FUNCTION_BLOCK BasicControlTS5 (* Basic Function Block Type *)
  (* Standard: 61499-2 *)
  (* Version 0.0, 6/17/2016, Andrei, nxtControl GmbH, Template *)
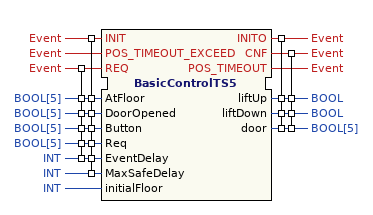
  EVENT_INPUT
    INIT WITH AtFloor, DoorOpened, Button, Req, EventDelay, MaxSafeDelay; (* Initialization Request *)
    POS_TIMEOUT_EXCEED;
    REQ WITH AtFloor, DoorOpened, Button, Req, EventDelay; (* Normal Execution Request *)
  END_EVENT
  EVENT_OUTPUT
    INITO WITH liftUp, liftDown, door; (* Initialization Confirm *)
    CNF WITH liftUp, liftDown, door; (* Execution Confirmation *)
    POS_TIMEOUT;
  END_EVENT
  VAR_INPUT
    AtFloor : ARRAY [0..4] OF BOOL; (* Input event qualifier *)
    DoorOpened : ARRAY [0..4] OF BOOL;
    Button : ARRAY [0..4] OF BOOL;
    Req : ARRAY [0..4] OF BOOL;
    EventDelay : INT;
    MaxSafeDelay : INT;
    initialFloor : INT := 2;
  END_VAR
  VAR_OUTPUT
    liftUp : BOOL;
    liftDown : BOOL; (* Output event qualifier *)
    door : ARRAY [0..4] OF BOOL;
  END_VAR
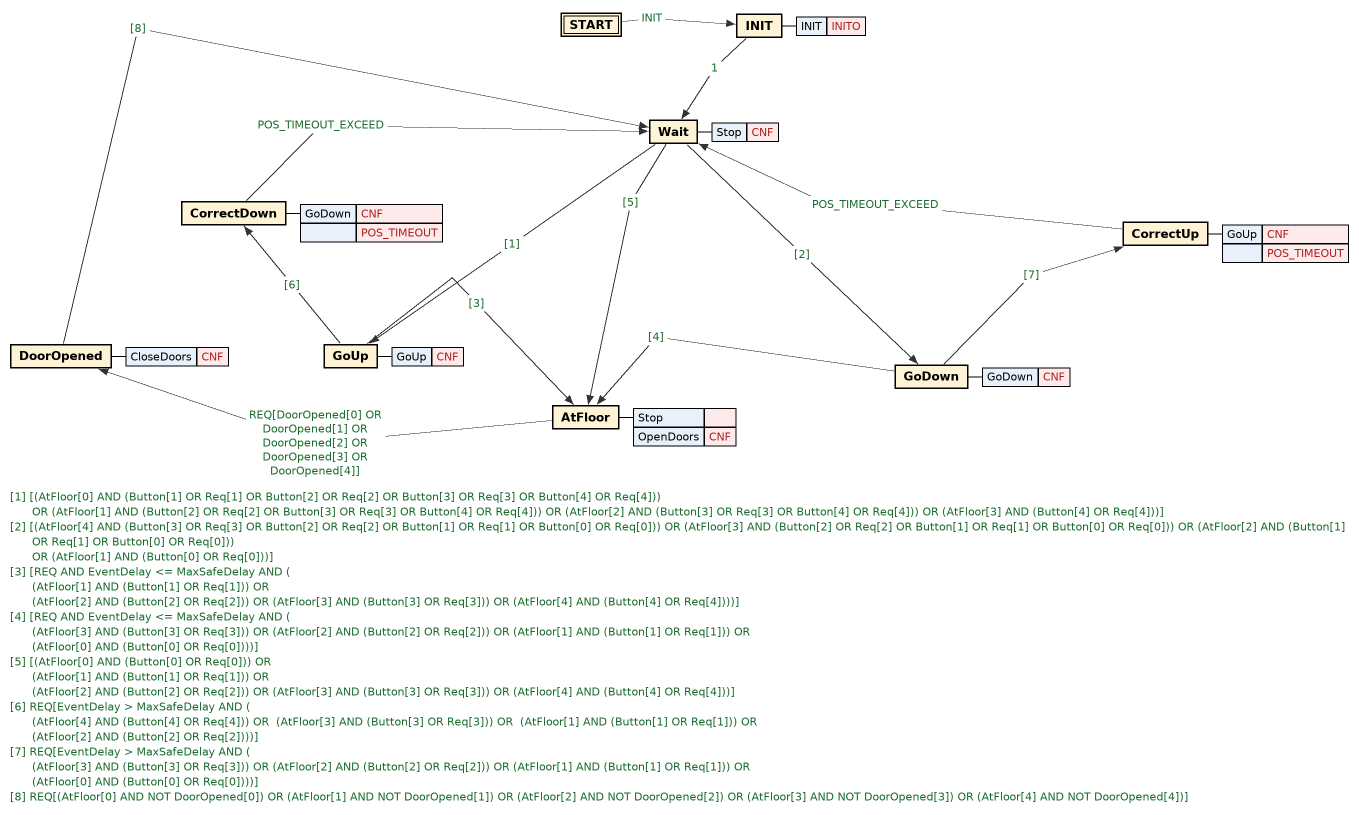
  EC_STATES
    START; (* Initial State *)
    INIT : INIT -> INITO; (* Initialization *)
    AtFloor : Stop, OpenDoors -> CNF;
    GoUp : GoUp -> CNF;
    Wait : Stop -> CNF;
    DoorOpened : CloseDoors -> CNF;
    GoDown : GoDown -> CNF;
    CorrectDown : GoDown -> CNF, -> POS_TIMEOUT;
    CorrectUp : GoUp -> CNF, -> POS_TIMEOUT;
  END_STATES
  EC_TRANSITIONS
    START TO INIT := INIT;
    INIT TO Wait := 1;
    GoUp TO AtFloor := [REQ AND EventDelay <= MaxSafeDelay AND ( (AtFloor[1] AND (Button[1] OR Req[1])) OR (AtFloor[2] AND (Button[2] OR Req[2])) OR (AtFloor[3] AND (Button[3] OR Req[3])) OR (AtFloor[4] AND (Button[4] OR Req[4])))];
    Wait TO AtFloor := [(AtFloor[0] AND (Button[0] OR Req[0])) OR (AtFloor[1] AND (Button[1] OR Req[1])) OR (AtFloor[2] AND (Button[2] OR Req[2])) OR (AtFloor[3] AND (Button[3] OR Req[3])) OR (AtFloor[4] AND (Button[4] OR Req[4]))];
    Wait TO GoUp := [(AtFloor[0] AND (Button[1] OR Req[1] OR Button[2] OR Req[2] OR Button[3] OR Req[3] OR Button[4] OR Req[4])) OR (AtFloor[1] AND (Button[2] OR Req[2] OR Button[3] OR Req[3] OR Button[4] OR Req[4])) OR (AtFloor[2] AND (Button[3] OR Req[3] OR Button[4] OR Req[4])) OR (AtFloor[3] AND (Button[4] OR Req[4]))];
    AtFloor TO DoorOpened := REQ[DoorOpened[0] OR DoorOpened[1] OR DoorOpened[2] OR DoorOpened[3] OR DoorOpened[4]];
    GoDown TO AtFloor := [REQ AND EventDelay <= MaxSafeDelay AND ( (AtFloor[3] AND (Button[3] OR Req[3])) OR (AtFloor[2] AND (Button[2] OR Req[2])) OR (AtFloor[1] AND (Button[1] OR Req[1])) OR (AtFloor[0] AND (Button[0] OR Req[0])))];
    GoUp TO CorrectDown := REQ[EventDelay > MaxSafeDelay AND ( (AtFloor[4] AND (Button[4] OR Req[4])) OR  (AtFloor[3] AND (Button[3] OR Req[3])) OR  (AtFloor[1] AND (Button[1] OR Req[1])) OR (AtFloor[2] AND (Button[2] OR Req[2])))];
    GoDown TO CorrectUp := REQ[EventDelay > MaxSafeDelay AND ( (AtFloor[3] AND (Button[3] OR Req[3])) OR (AtFloor[2] AND (Button[2] OR Req[2])) OR (AtFloor[1] AND (Button[1] OR Req[1])) OR (AtFloor[0] AND (Button[0] OR Req[0])))];
    Wait TO GoDown := [(AtFloor[4] AND (Button[3] OR Req[3] OR Button[2] OR Req[2] OR Button[1] OR Req[1] OR Button[0] OR Req[0])) OR (AtFloor[3] AND (Button[2] OR Req[2] OR Button[1] OR Req[1] OR Button[0] OR Req[0])) OR (AtFloor[2] AND (Button[1] OR Req[1] OR Button[0] OR Req[0])) OR (AtFloor[1] AND (Button[0] OR Req[0]))];
    DoorOpened TO Wait := REQ[(AtFloor[0] AND NOT DoorOpened[0]) OR (AtFloor[1] AND NOT DoorOpened[1]) OR (AtFloor[2] AND NOT DoorOpened[2]) OR (AtFloor[3] AND NOT DoorOpened[3]) OR (AtFloor[4] AND NOT DoorOpened[4])];
    CorrectUp TO Wait := POS_TIMEOUT_EXCEED;
    CorrectDown TO Wait := POS_TIMEOUT_EXCEED;
  END_TRANSITIONS
  ALGORITHM INIT IN ST: (* Initialization algorithm *)
liftDown := FALSE;
liftUp := FALSE;
  END_ALGORITHM
  ALGORITHM GoDown IN ST:
liftDown := TRUE;
liftUp := FALSE;
  END_ALGORITHM
  ALGORITHM Stop IN ST:
liftDown := FALSE;
liftUp := FALSE;
  END_ALGORITHM
  ALGORITHM GoUp IN ST: (* new algorithm *)
;
liftUp :=TRUE;
liftDown := FALSE;
  END_ALGORITHM
  ALGORITHM OpenDoors IN ST: (* new algorithm *)
door[0] := AtFloor[0];
door[1] := AtFloor[1];
door[2] := AtFloor[2];
door[3] := AtFloor[3];
door[4] := AtFloor[4];
  END_ALGORITHM
  ALGORITHM CloseDoors IN ST: (* new algorithm *)
door[0] := FALSE;
door[1] := FALSE;
door[2] := FALSE;
door[3] := FALSE;
door[4] := FALSE;
  END_ALGORITHM
END_FUNCTION_BLOCK
